PROGRAM AxisServoCtrl_Arm1
VAR

	fbArm1VertServoMasterController 	: fbV2_ServoMasterController;
	fbArm1HorzServoMasterController 	: fbV2_ServoMasterController;

	iArm1VertStepNumber				: INT;
	iArm1HorzStepNumber				: INT;

	bArm1MCPSOV					: BOOL;
	bArm1MCPSOH					: BOOL;

	bVertDiagBusy					: BOOL;
	bHorzDiagBusy					: BOOL;

	iVertClass3Diag					: INT;
	iHorzClass3Diag					: INT;

	iVertstAX5000C1D					: ST_AX5000_C1D;
	iHorzstAX5000C1D				: ST_AX5000_C1D;

END_VAR

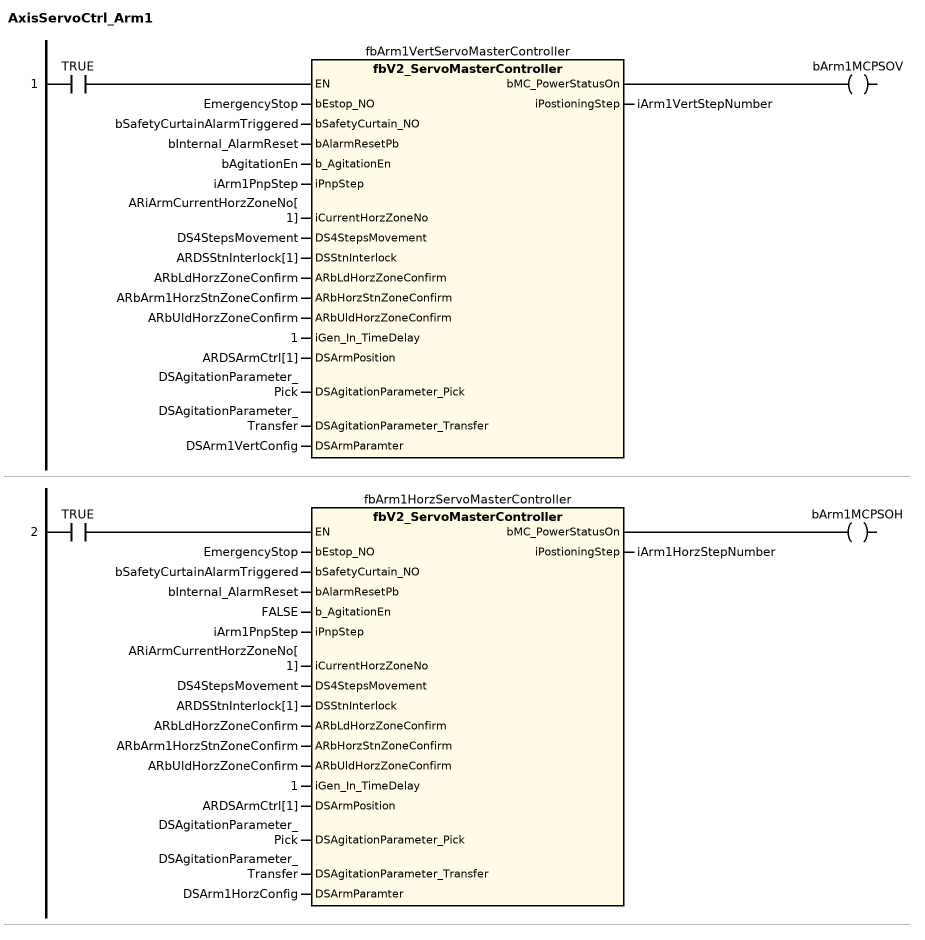
// NETWORK 1
fbArm1VertServoMasterController(
    bEstop_NO := EmergencyStop,
    bSafetyCurtain_NO := bSafetyCurtainAlarmTriggered,
    bAlarmResetPb := bInternal_AlarmReset,
    b_AgitationEn := bAgitationEn,
    iPnpStep := iArm1PnpStep,
    iCurrentHorzZoneNo := ARiArmCurrentHorzZoneNo[1],
    DS4StepsMovement := DS4StepsMovement,
    DSStnInterlock := ARDSStnInterlock[1],
    ARbLdHorzZoneConfirm := ARbLdHorzZoneConfirm,
    ARbHorzStnZoneConfirm := ARbArm1HorzStnZoneConfirm,
    ARbUldHorzZoneConfirm := ARbUldHorzZoneConfirm,
    iGen_In_TimeDelay := 1,
    DSArmPosition := ARDSArmCtrl[1],
    DSAgitationParameter_Pick := DSAgitationParameter_Pick,
    DSAgitationParameter_Transfer := DSAgitationParameter_Transfer,
    DSArmParamter := DSArm1VertConfig,
    iPostioningStep => iArm1VertStepNumber); // fbV2_ServoMasterController
bArm1MCPSOV := fbArm1VertServoMasterController.bMC_PowerStatusOn;

// NETWORK 2
fbArm1HorzServoMasterController(
    bEstop_NO := EmergencyStop,
    bSafetyCurtain_NO := bSafetyCurtainAlarmTriggered,
    bAlarmResetPb := bInternal_AlarmReset,
    b_AgitationEn := FALSE,
    iPnpStep := iArm1PnpStep,
    iCurrentHorzZoneNo := ARiArmCurrentHorzZoneNo[1],
    DS4StepsMovement := DS4StepsMovement,
    DSStnInterlock := ARDSStnInterlock[1],
    ARbLdHorzZoneConfirm := ARbLdHorzZoneConfirm,
    ARbHorzStnZoneConfirm := ARbArm1HorzStnZoneConfirm,
    ARbUldHorzZoneConfirm := ARbUldHorzZoneConfirm,
    iGen_In_TimeDelay := 1,
    DSArmPosition := ARDSArmCtrl[1],
    DSAgitationParameter_Pick := DSAgitationParameter_Pick,
    DSAgitationParameter_Transfer := DSAgitationParameter_Transfer,
    DSArmParamter := DSArm1HorzConfig,
    iPostioningStep => iArm1HorzStepNumber); // fbV2_ServoMasterController
bArm1MCPSOH := fbArm1HorzServoMasterController.bMC_PowerStatusOn;

END_PROGRAM

(* stored: Version 1.1.0.1, ProductVersion 3.1.4024.12
   POU AxisServoCtrl_Arm1: Id {96edea8f-7050-4049-9c9d-8d2b4af3d590}, SpecialFunc None *)
